FUNCTION_BLOCK FB_LogOnEdge
VAR_INPUT
   Event : BOOL; // look for edge here to log.
   Message : T_MaxString; // message
   LogSeverity : E_LogSeverity; // severity
   EventFallingEdge : BOOL := FALSE; // TRUE for falling edge, FALSE for rising edge.
END_VAR
VAR_OUTPUT
   Q : BOOL;
END_VAR
VAR
   rt : R_TRIG;
   ft : F_TRIG;
END_VAR
VAR_TEMP
   logNow : BOOL;
END_VAR

rt(CLK := Event);
ft(CLK := Event);

Q := SEL(EventFallingEdge, rt.Q, ft.Q);

IF Q THEN

   CASE LogSeverity OF

      E_LogSeverity.Info:
         F_LogInfo(Message);

      E_LogSeverity.Warning:
         F_LogWarning(Message);

      E_LogSeverity.Error:
         F_LogError(Message);
   ELSE

      F_LogError(
         CONCAT(
            'Error in FB_LogOnEdge, Logseverity incorrect. Log Message for event is : ',
            Message
         )
      );

   END_CASE

END_IF

END_FUNCTION_BLOCK

(* stored: Version 1.1.0.1, ProductVersion 3.1.4026.12
   POU FB_LogOnEdge: Id {7a4e7629-be67-098c-3b9d-bcb39afe4228}, SpecialFunc None *)
